{attribute 'qualified_only'}
{attribute 'strict'}
{attribute 'to_string'}
TYPE E_Motion :
(
	Sine,
	Ramp
);
END_TYPE

(* stored: Version 1.1.0.1
   DUT E_Motion: Id {c3639952-caae-49ba-bea6-50f8226af1ab} *)
